INTERFACE ITcoResultsData

END_INTERFACE

(* stored: Version 1.1.0.1, ProductVersion 3.1.4024.12
   Itf ITcoResultsData: Id {46ba482a-b036-0503-2755-d75f19774c6a} *)
